INTERFACE I_Sensor

PROPERTY Calibrado : BOOL
GET
END_GET
END_PROPERTY

METHOD Calibrar
END_METHOD

PROPERTY Consigna : REAL
SET
END_SET
END_PROPERTY


METHOD Descalibrar
END_METHOD

METHOD LeerValor : INT
END_METHOD

PROPERTY Temperatura : REAL
GET
END_GET
END_PROPERTY

END_INTERFACE

(* stored: Version 1.1.0.1, ProductVersion 3.1.4024.12
   Itf I_Sensor: Id {7958397f-48a8-454b-a010-e0414fe583b5}
   Property Calibrado: Id {8abbaf26-ce96-4b0f-8e8d-9725437ad921}
   Get Get: Id {1eb2e9ac-1877-4b17-9c46-f99cd39d7ba0}
   Method Calibrar: Id {7f96ac36-f28a-4f3e-a22b-092e448c5536}
   Property Consigna: Id {821330b5-8774-4b25-9254-6d215d35ad0e}
   Set Set: Id {4313bf85-918e-4f5a-9c86-520a431b4978}
   Method Descalibrar: Id {8931e251-8ce4-45d1-b61d-04a569c5ea3a}
   Method LeerValor: Id {ad9fd777-b86e-4466-948f-7e3fc3051ec9}
   Property Temperatura: Id {a2fe7ee0-b9bf-4f16-a423-09fd1413b014}
   Get Get: Id {cf328966-d649-4268-9431-0081cc38ea31} *)
